FUNCTION_BLOCK START_STOP_CONTROLLER (* Composite Function Block Type *)
  (* Standard: 61499-2 *)
  (* Version 1.0, 2019-04-12, adeel *)
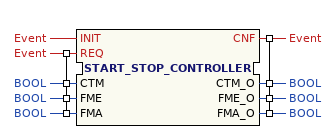
  EVENT_INPUT
    INIT; (* Initialization Request *)
    REQ WITH CTM, FME, FMA; (* Normal Execution Request *)
  END_EVENT
  EVENT_OUTPUT
    CNF WITH CTM_O, FME_O, FMA_O; (* Execution Confirmation *)
  END_EVENT
  VAR_INPUT
    CTM : BOOL;
    FME : BOOL;
    FMA : BOOL;
  END_VAR
  VAR_OUTPUT
    CTM_O : BOOL;
    FME_O : BOOL;
    FMA_O : BOOL;
  END_VAR
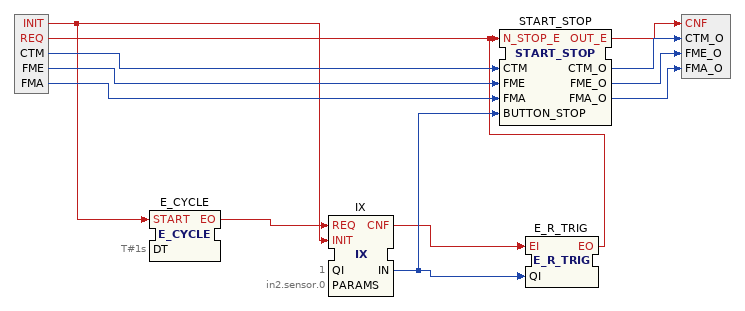
  FBS
    START_STOP : START_STOP;
    IX : IX(QI := 1, PARAMS := in2.sensor.0);
    E_CYCLE : E_CYCLE(DT := T#1s);
    E_R_TRIG : E_R_TRIG;
  END_FBS
  EVENT_CONNECTIONS
    E_CYCLE.EO TO IX.REQ;
    INIT TO IX.INIT;
    INIT TO E_CYCLE.START;
    REQ TO START_STOP.N_STOP_E;
    START_STOP.OUT_E TO CNF;
    IX.CNF TO E_R_TRIG.EI;
    E_R_TRIG.EO TO START_STOP.N_STOP_E;
  END_CONNECTIONS
  DATA_CONNECTIONS
    IX.IN TO START_STOP.BUTTON_STOP;
    CTM TO START_STOP.CTM;
    FME TO START_STOP.FME;
    FMA TO START_STOP.FMA;
    START_STOP.CTM_O TO CTM_O;
    START_STOP.FME_O TO FME_O;
    START_STOP.FMA_O TO FMA_O;
    IX.IN TO E_R_TRIG.QI;
  END_CONNECTIONS
END_FUNCTION_BLOCK
